% RSLogix 500 project I2P Hands-On 3 - Alexander.RSS, saved by version 10.00.00.00 %
PROJECT "ML05B"    % processor: Bul.1763 MicroLogix 1100 Series B %

PROGRAM FILES
  LAD 2   13 rungs

DATA FILES
  O0 OUTPUT  4 elements
  I1 INPUT  6 elements
  S2 STATUS  66 elements
  B3 BINARY  1 elements
  T4 TIMER  1 elements
  C5 COUNTER  1 elements
  R6 CONTROL  1 elements
  N7 INTEGER  1 elements
  F8 FLOAT  1 elements

LADDER 2
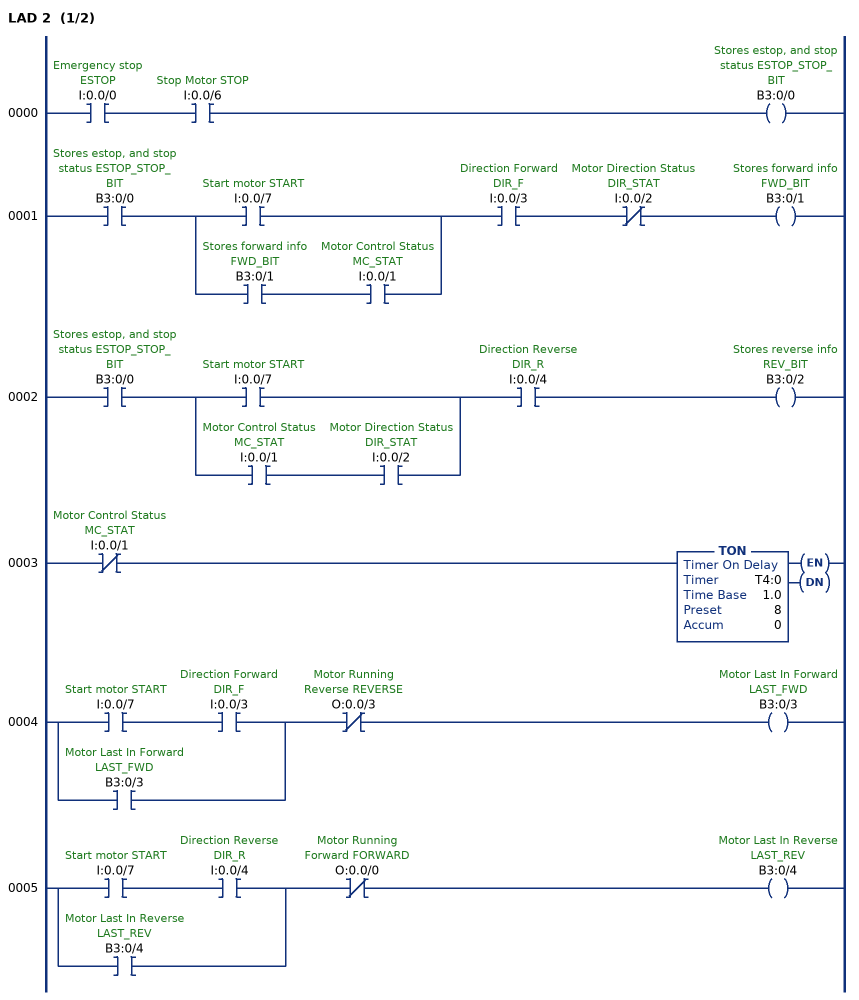
% Rung: 0 %
SOR XIC I:0.0/0 XIC I:0.0/6 OTE B3:0/0 EOR
%   I:0.0/0  ESTOP  "Emergency stop" %
%   I:0.0/6  STOP  "Stop Motor" %
%   B3:0/0  ESTOP_STOP_BIT  "Stores estop, and stop status" %
% Rung: 1 %
SOR XIC B3:0/0 BST XIC I:0.0/7 NXB XIC B3:0/1 XIC I:0.0/1 BND XIC I:0.0/3 XIO I:0.0/2 OTE B3:0/1 EOR
%   B3:0/0  ESTOP_STOP_BIT  "Stores estop, and stop status" %
%   I:0.0/7  START  "Start motor" %
%   B3:0/1  FWD_BIT  "Stores forward info" %
%   I:0.0/1  MC_STAT  "Motor Control Status" %
%   I:0.0/3  DIR_F  "Direction Forward" %
%   I:0.0/2  DIR_STAT  "Motor Direction Status" %
% Rung: 2 %
SOR XIC B3:0/0 BST XIC I:0.0/7 NXB XIC I:0.0/1 XIC I:0.0/2 BND XIC I:0.0/4 OTE B3:0/2 EOR
%   B3:0/0  ESTOP_STOP_BIT  "Stores estop, and stop status" %
%   I:0.0/7  START  "Start motor" %
%   I:0.0/1  MC_STAT  "Motor Control Status" %
%   I:0.0/2  DIR_STAT  "Motor Direction Status" %
%   I:0.0/4  DIR_R  "Direction Reverse" %
%   B3:0/2  REV_BIT  "Stores reverse info" %
% Rung: 3 %
SOR XIO I:0.0/1 TON T4:0 1.0 8 0 EOR
%   I:0.0/1  MC_STAT  "Motor Control Status" %
% Rung: 4 %
SOR BST XIC I:0.0/7 XIC I:0.0/3 NXB XIC B3:0/3 BND XIO O:0.0/3 OTE B3:0/3 EOR
%   I:0.0/7  START  "Start motor" %
%   I:0.0/3  DIR_F  "Direction Forward" %
%   B3:0/3  LAST_FWD  "Motor Last In Forward" %
%   O:0.0/3  REVERSE  "Motor Running Reverse" %
% Rung: 5 %
SOR BST XIC I:0.0/7 XIC I:0.0/4 NXB XIC B3:0/4 BND XIO O:0.0/0 OTE B3:0/4 EOR
%   I:0.0/7  START  "Start motor" %
%   I:0.0/4  DIR_R  "Direction Reverse" %
%   B3:0/4  LAST_REV  "Motor Last In Reverse" %
%   O:0.0/0  FORWARD  "Motor Running Forward" %

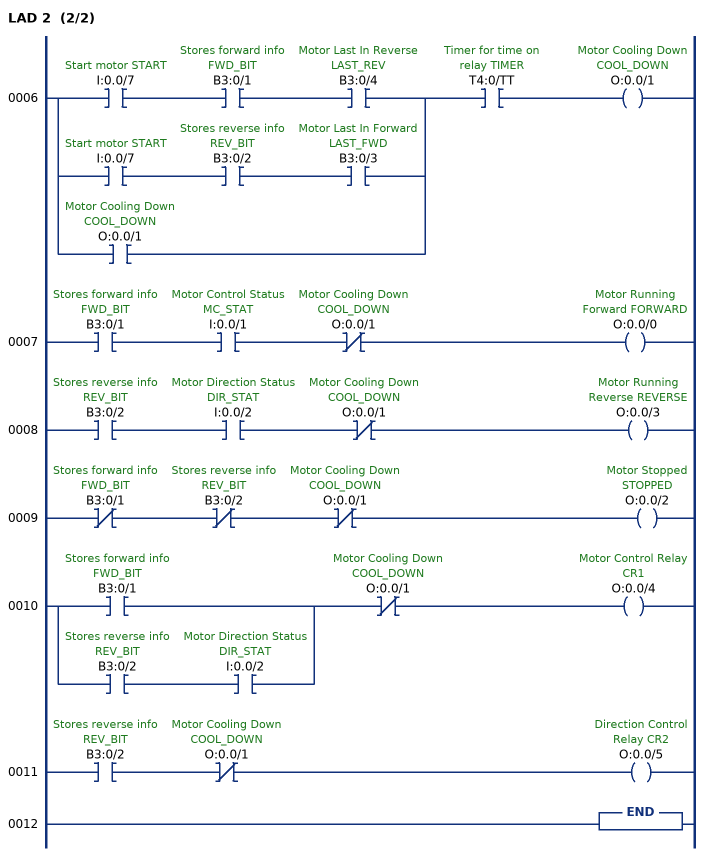
% Rung: 6 %
SOR BST XIC I:0.0/7 XIC B3:0/1 XIC B3:0/4 NXB BST XIC I:0.0/7 XIC B3:0/2 XIC B3:0/3 NXB XIC O:0.0/1 BND BND XIC T4:0/TT OTE O:0.0/1 EOR
%   I:0.0/7  START  "Start motor" %
%   B3:0/1  FWD_BIT  "Stores forward info" %
%   B3:0/4  LAST_REV  "Motor Last In Reverse" %
%   B3:0/2  REV_BIT  "Stores reverse info" %
%   B3:0/3  LAST_FWD  "Motor Last In Forward" %
%   O:0.0/1  COOL_DOWN  "Motor Cooling Down" %
%   T4:0/TT  TIMER  "Timer for time on relay" %
% Rung: 7 %
SOR XIC B3:0/1 XIC I:0.0/1 XIO O:0.0/1 OTE O:0.0/0 EOR
%   B3:0/1  FWD_BIT  "Stores forward info" %
%   I:0.0/1  MC_STAT  "Motor Control Status" %
%   O:0.0/1  COOL_DOWN  "Motor Cooling Down" %
%   O:0.0/0  FORWARD  "Motor Running Forward" %
% Rung: 8 %
SOR XIC B3:0/2 XIC I:0.0/2 XIO O:0.0/1 OTE O:0.0/3 EOR
%   B3:0/2  REV_BIT  "Stores reverse info" %
%   I:0.0/2  DIR_STAT  "Motor Direction Status" %
%   O:0.0/1  COOL_DOWN  "Motor Cooling Down" %
%   O:0.0/3  REVERSE  "Motor Running Reverse" %
% Rung: 9 %
SOR XIO B3:0/1 XIO B3:0/2 XIO O:0.0/1 OTE O:0.0/2 EOR
%   B3:0/1  FWD_BIT  "Stores forward info" %
%   B3:0/2  REV_BIT  "Stores reverse info" %
%   O:0.0/1  COOL_DOWN  "Motor Cooling Down" %
%   O:0.0/2  STOPPED  "Motor Stopped" %
% Rung: 10 %
SOR BST XIC B3:0/1 NXB XIC B3:0/2 XIC I:0.0/2 BND XIO O:0.0/1 OTE O:0.0/4 EOR
%   B3:0/1  FWD_BIT  "Stores forward info" %
%   B3:0/2  REV_BIT  "Stores reverse info" %
%   I:0.0/2  DIR_STAT  "Motor Direction Status" %
%   O:0.0/1  COOL_DOWN  "Motor Cooling Down" %
%   O:0.0/4  CR1  "Motor Control Relay" %
% Rung: 11 %
SOR XIC B3:0/2 XIO O:0.0/1 OTE O:0.0/5 EOR
%   B3:0/2  REV_BIT  "Stores reverse info" %
%   O:0.0/1  COOL_DOWN  "Motor Cooling Down" %
%   O:0.0/5  CR2  "Direction Control Relay" %
% Rung: 12 %
SOR END EOR

OTHER DOCUMENTED ADDRESSES
  B3:0/5  C  "Motor is cooling do"

DATA TABLE (non-zero values as saved)
DATA B3
% B3:0 % 0X0001
DATA T4
% .PRE .ACC %
% T4:0 % 8 0
